Staubli VAL3: onEnterEvent.pgx

program onEnterEvent()
  local num l_nResult
  local string l_sMessage
begin
  if sEvent!=""

    if  save:nBoxType==1
      set:bWizard=false
      call set:editSmlData(sEvent,l_nResult)
      call language2:message(l_sMessage,4)
      call use:timerDialog(l_sMessage,0)
      call set:onSave()
    elseIf save:nBoxType==2
      set:bWizard=false
      call set:editBigData(sEvent,l_nResult)
      call language2:message(l_sMessage,4)
      call use:timerDialog(l_sMessage,0)
      call set:onSave()
    endIf
  endIf
end
